// TwinCAT 3 PLC project TcOpenPlc
// Title: TcOpenPlc
// Company: TcOpenGroup
// ProjectVersion: 0.0.0.1
// ProgramVersion: 3.1.4023.0
// libraries:
//   Tc2_Standard, * (Beckhoff Automation GmbH)
//   Tc2_System, * (Beckhoff Automation GmbH)
//   Tc3_Module, * (Beckhoff Automation GmbH)
//   TcoCore, 0.4.2.718 (Vortex.Library)
//   TcoData, 0.4.2.718 (Vortex.Library)
//   TcoDrivesBeckhoff, 0.4.2.718 (Vortex.Library)
//   TcoElements, 0.4.2.718 (Vortex.Library)
//   TcoIoBeckhoff, 0.4.2.718 (Vortex.Library)
//   TcoPneumatics, 0.4.2.718 (Vortex.Library)
// project tree:
//   / PlcTask.TcTTO (not stored)
//   POUs/ MAIN.TcPOU, SimpleContext.TcPOU
//   POUs/ST1/ IO.TcGVL, ST001.TcPOU
// real-time tasks:
//   TASK PlcTask: cycle T#10ms, priority 20, ADS port 350

// ---- POUs/ST1/IO.TcGVL
{attribute 'qualified_only'}
VAR_GLOBAL
	iCH_1 AT %I* : BOOL;
	iCH_2 AT %I* : BOOL;
	iCH_3 AT %I* : BOOL;
	iCH_4 AT %I* : BOOL;
	iCH_5 AT %I* : BOOL;
	iCH_6 AT %I* : BOOL;
	iCH_7 AT %I* : BOOL;
	iCH_8 AT %I* : BOOL;


	qCH_1 AT %Q* : BOOL;
	qCH_2 AT %Q* : BOOL;
	qCH_3 AT %Q* : BOOL;
	qCH_4 AT %Q* : BOOL;
	qCH_5 AT %Q* : BOOL;
	qCH_6 AT %Q* : BOOL;
	qCH_7 AT %Q* : BOOL;
	qCH_8 AT %Q* : BOOL;	
END_VAR

// ---- POUs/MAIN.TcPOU
PROGRAM MAIN
VAR
	_simpleContext : SimpleContext;
END_VAR

_simpleContext.Run();

END_PROGRAM

// ---- POUs/SimpleContext.TcPOU
FUNCTION_BLOCK SimpleContext EXTENDS TcoCore.TcoContext
VAR
	_st001 : ST001(THIS^);
	_messenger : TcoCore.TcoMessenger(THIS^); 
	_angelos : ARRAY[0..10] OF TcoCore.TcoMessenger(THIS^);
END_VAR

(*~
	<docu>
		<summary>
			Main method of the TcoContext. This is the entry point of any control logic that belongs to this context. 
			The call of this method is ensured by calling the <c>InstanceName.Run()</c> method, and it must not be called explicitly.
			This method is abstract, and it must be overridden in derived block.
		</summary>
	</docu>
~*)
METHOD PROTECTED  Main
THIS^.Environment.Messaging.MessageDigestMethod := eMessageDigestMethod.CRC32;
THIS^.Environment.Messaging.MessengerLoggingMethod := eMessengerLogMethod.OnEventRisen;

_messenger.Info('This is an info message');
_messenger.Error('This is an error message');
_messenger.Critical('This is an critical message 1111');

_st001();




























//IF(THIS^._startCycleCount MOD 10 = 0) THEN
//	Logger.Push('This is a log entry', eMessageCategory.Trace);
//END_IF;	

//IF(THIS^._startCycleCount MOD 125 = 0) THEN
//	Logger.Push('This is a log entry', eMessageCategory.Info);
//END_IF;	

//IF(THIS^._startCycleCount MOD 400 = 0) THEN
//	Logger.Push('This is a log entry', eMessageCategory.Warning);
//END_IF;	

//IF(THIS^._startCycleCount MOD 2000 = 0) THEN
//	Logger.Push('This is a log entry', eMessageCategory.Error);
//END_IF;
END_METHOD

END_FUNCTION_BLOCK

// ---- POUs/ST1/ST001.TcPOU
FUNCTION_BLOCK ST001 EXTENDS TcoCore.TcoObject
VAR
	_piston : TcoPneumatics.TcoCylinder(THIS^);
	_state : INT;
END_VAR

_piston(inoAtHomePos:= IO.iCH_1, inoAtWorkPos:= IO.iCH_2, inoToHomePos:= IO.qCH_1, inoToWorkPos:=IO.qCH_2);

CASE _state OF
	0:
		IF(_piston.MoveToHome().Done) THEN
			_state := 10;
		END_IF
	10:
		IF(_piston.MoveToWork().Done) THEN
			_state := 20;
		END_IF
	20:
		_state := 0;
END_CASE


Messenger.Trace(CONCAT('Running state: ', INT_TO_STRING(_state)));

END_FUNCTION_BLOCK
